// TIA Portal V20 export
DATA_BLOCK "Config"   // DB195
// stored: MemoryReserve 100, Namespace Unit1
   VAR
      unit : "LAF_typeUnitConfiguration";   // Configuration of Unit Parameters
      stateMachine : "LUC_typeStateMachineConfiguration";
      signalStack : "LUC_typeSignalStackConfiguration";
      remoteCtrlOpcUa : "LUC_typeRemoteCtrlConfiguration";
      stateModeManager { ExternalAccessible := 'False'; ExternalVisible := 'False'; ExternalWritable := 'False'} : "LPMLV2022_typeConfiguration";   // Do not change. Can be configured through stateMachineConfiguration
      cmFFU_LIU117 : "LER_typeLIU117Configuration";
      sleep { S7_SetPoint := 'True'} : "LER_typeSleepModeParameter";
      "========Communication========" : Bool;
      BA030 : "LER_typeCommunicationConfiguration";
      BA040 : "LER_typeCommunicationConfiguration";
      BA100 { S7_SetPoint := 'True'} : "LER_typeCommunicationConfiguration";
      CoveyorA : "LER_typeCommunicationConfiguration";
   END_VAR
BEGIN
   unit.referenceDesignator.relative := WSTRING#'U2';
   stateMachine.enableModes.noMode := true;
   cmFFU_LIU117.MB_Comm_Load.PORT := 514;
   cmFFU_LIU117.MB_Comm_Load.BAUD := 9600;
   BA030.SEND.connectionId := 16#162;
   BA030.SEND.rid := 16#16;
   BA030.RCV.connectionId := 16#162;
   BA030.RCV.rid := 16#15;
   BA040.SEND.connectionId := 16#172;
   BA040.SEND.rid := 16#26;
   BA040.RCV.connectionId := 16#172;
   BA040.RCV.rid := 16#25;
   BA100.SEND.connectionId := 16#182;
   BA100.SEND.rid := 16#31;
   BA100.RCV.connectionId := 16#182;
   BA100.RCV.rid := 16#32;
   CoveyorA.SEND.connectionId := 16#172;
   CoveyorA.SEND.rid := 16#26;
   CoveyorA.RCV.connectionId := 16#172;
   CoveyorA.RCV.rid := 16#25;
END_DATA_BLOCK
